// TwinCAT 3 PLC project ExamplePlc
// Company: Sensata Technologies Mechanization
// ProgramVersion: 3.1.4023.0
// libraries:
//   Sensata_Common, * (Sensata Technologies)
//   Sensata_PressureTransducers, * (Sensata Technologies)
//   Sensata_Utilities, * (Sensata Technologies)
//   Tc2_Standard, * (Beckhoff Automation GmbH)
//   Tc2_System, * (Beckhoff Automation GmbH)
//   Tc2_Utilities, * (Beckhoff Automation GmbH)
//   Tc3_Module, * (Beckhoff Automation GmbH)
// project tree:
//   0 Program/ PRG_Main.TcPOU
//   1 Module/0 Machines/ FB_ExampleMachine.TcPOU (not stored)
//   1 Module/1 Stations/ FB_ExampleStation.TcPOU (not stored)
//   1 Module/2 Devices/ FB_ExampleDevice.TcPOU (not stored)
//   / TASK_Main.TcTTO (not stored)
// real-time tasks:
//   TASK TASK_Main: cycle T#10ms, priority 20, ADS port 350

// ---- 0 Program/PRG_Main.TcPOU
PROGRAM PRG_Main
VAR
	bTestInput: BOOL;
	bTestOutput: BOOL;
	fbMachine: FB_ExampleMachine;
	fbStation1: FB_ExampleStation;
	fbStation2: FB_ExampleStation;
	fbStation3: FB_ExampleStation;
	fbStation4: FB_ExampleStation;
	bStart: BOOL;
	bAbort: BOOL;
	bReset: BOOL;
	bStop: BOOL;
	bSuspend: BOOL;
	fbDevice1: FB_ExampleDevice;
	fbDevice2: FB_ExampleDevice;
	fbDevice3: FB_ExampleDevice;
	fbDevice4: FB_ExampleDevice;
	bPoweredOn: BOOL;
//	FB_AdsDeviceAPI_0: FB_AdsDeviceAPI;
	FB_AdsDeviceAPI_0 : FB_AdsCommandRouter;
	bConnectToAlicatAbs: BOOL;
	bRes_AlicatAbsConnected: BOOL;
	bTestADSServer: BOOL;
	strTarget: T_MaxString;
	strCommand: T_MaxString;
	arrParams: T_ApiMethodParameters;
	MyResults: T_MaxString;
	bInterfaceTest : BOOL;
	bDisconnectFromAlicatAbs: BOOL;
	bRes_AlicatAbsDisConnected: BOOL;
	bGetPressure: BOOL;
	bGetPressureSuccessful: BOOL;
	bGetAlicatData: BOOL;
	bGetAlicatDataSuccessful: BOOL;
	bLockDisplay: BOOL;
	bLockDisplaySuccessful: BOOL;
	bUnlockDisplay: BOOL;
	bUnlockDisplaySuccessful: BOOL;
	AlicatAbsolutePressureTransducer_1: FB_AbsolutePressureTransducer;
END_VAR

bTestOutput := bTestInput;

A_Machine();
//A_Station1();
//A_Station2();
//A_Station3();
//A_Station4();
//bInterfaceTest := MyLaser1.fbApi.P_bDeviceInterfaceBusy;



IF bConnectToAlicatAbs THEN
	bRes_AlicatAbsConnected := AlicatAbsolutePressureTransducer_1.M_Connect();
	IF bRes_AlicatAbsConnected THEN
		bConnectToAlicatAbs := FALSE;
	ELSIF AlicatAbsolutePressureTransducer_1.P_bError THEN
		bConnectToAlicatAbs := FALSE;
		AlicatAbsolutePressureTransducer_1.M_ClearError();
	END_IF
END_IF

IF bDisconnectFromAlicatAbs THEN
	bRes_AlicatAbsDisConnected := AlicatAbsolutePressureTransducer_1.M_Disconnect();
	IF bRes_AlicatAbsConnected THEN
		bDisconnectFromAlicatAbs := FALSE;
	ELSIF AlicatAbsolutePressureTransducer_1.P_bError THEN
		bDisconnectFromAlicatAbs := FALSE;
		AlicatAbsolutePressureTransducer_1.M_ClearError();
	END_IF
END_IF

IF bGetPressure THEN
	bGetPressureSuccessful := AlicatAbsolutePressureTransducer_1.M_GetPressure();
	IF bGetPressureSuccessful THEN
		bGetPressure := FALSE;
	ELSIF AlicatAbsolutePressureTransducer_1.P_bError THEN
		bGetPressure := FALSE;
		AlicatAbsolutePressureTransducer_1.M_ClearError();
	END_IF
END_IF

IF bGetAlicatData THEN
	bGetAlicatDataSuccessful := AlicatAbsolutePressureTransducer_1.M_GetAlicatData();
	IF bGetAlicatDataSuccessful THEN
		bGetAlicatData := FALSE;
	ELSIF AlicatAbsolutePressureTransducer_1.P_bError THEN
		bGetAlicatData := FALSE;
		AlicatAbsolutePressureTransducer_1.M_ClearError();
	END_IF
END_IF

IF bLockDisplay THEN
	bLockDisplaySuccessful := AlicatAbsolutePressureTransducer_1.M_LockDisplay();
	IF bLockDisplaySuccessful THEN
		bLockDisplay := FALSE;
	ELSIF AlicatAbsolutePressureTransducer_1.P_bError THEN
		bLockDisplay := FALSE;
		AlicatAbsolutePressureTransducer_1.M_ClearError();
	END_IF
END_IF

IF bUnlockDisplay THEN
	bUnlockDisplaySuccessful := AlicatAbsolutePressureTransducer_1.M_UnlockDisplay();
	IF bUnlockDisplaySuccessful THEN
		bUnlockDisplay := FALSE;
	ELSIF AlicatAbsolutePressureTransducer_1.P_bError THEN
		bUnlockDisplay := FALSE;
		AlicatAbsolutePressureTransducer_1.M_ClearError();
	END_IF
END_IF


//IF bConnectToLaserMarker THEN
//	bRes_LaserConnected := MyLaser1.M_Connect();
//	IF bRes_LaserConnected THEN
//	//Add some timer based logic to do error handling.
//		bConnectToLaserMarker := FALSE;
//	ELSIF MyLaser1.P_bError THEN
//		bConnectToLaserMarker := FALSE;
//		MyLaser1.M_ClearError();
//	END_IF
//END_IF


//IF bDisconnectFromLaserMarker THEN
//	bRes_LaserDisconnected := MyLaser1.M_Disconnect();
//	IF bRes_LaserDisconnected THEN
//		bDisconnectFromLaserMarker := FALSE;
//	ELSIF MyLaser1.P_bError THEN
//		bDisconnectFromLaserMarker := FALSE;
//		MyLaser1.M_ClearError();
//	END_IF
//END_IF


//IF bPeakCurrentProgramInLaser THEN
//	bRes_PeakCurrentProgramInLaser := MyLaser1.M_PeakCurrentProgram();
//	IF bRes_PeakCurrentProgramInLaser THEN
//		bPeakCurrentProgramInLaser := FALSE;
//	ELSIF MyLaser1.P_bError THEN
//		bPeakCurrentProgramInLaser := FALSE;
//		MyLaser1.M_ClearError();
//	END_IF
//END_IF


//IF bSendProgramToLaser THEN
//	bRes_SendProgramtoLaser := MyLaser1.M_SendProgramtoLaser(filepath,LaserMemoryLocation);
//	IF bRes_SendProgramtoLaser THEN
//		bSendProgramToLaser := FALSE;
//	ELSIF MyLaser1.P_bError THEN
//		bSendProgramToLaser := FALSE;
//		MyLaser1.M_ClearError();
//	END_IF
//END_IF

//IF bSaveCurrentLaserProgramtoPC THEN
//	bRes_SaveCurrentLaserProgramtoPC := MyLaser1.M_SaveCurrentLaserProgramtoPC(LaserProgramFolderPath, out_bool_SaveProgramToPC_Success => SaveCurrentLaserProgramToPCSuccess);
//	IF bRes_SaveCurrentLaserProgramtoPC THEN
////		SaveCurrentLaserProgramToPCSuccess := MyLaser1
//		bSaveCurrentLaserProgramtoPC := FALSE;
//	ELSIF MyLaser1.P_bError THEN
//		bSaveCurrentLaserProgramtoPC := FALSE;
//		MyLaser1.M_ClearError();
//	END_IF
//END_IF

//IF bStartMarking THEN
//	bRes_StartMarking := MyLaser1.M_StartMarking();
//	IF bRes_StartMarking THEN
//		bStartMarking := FALSE;
//	ELSIF MyLaser1.P_bError THEN
//		bStartMarking := FALSE;
//		MyLaser1.M_ClearError();
//	END_IF
//END_IF

//IF bStopMarking THEN
//	bRes_StopMarking := MyLaser1.M_StopMarking();
//	IF bRes_StopMarking THEN
//		bStopMarking := FALSE;
//	ELSIF MyLaser1.P_bError THEN
//		bStopMarking := FALSE;
//		MyLaser1.M_ClearError();
//	END_IF
//END_IF

//IF bClearLaserErrors THEN
//	bRes_ClearLaserErrors := MyLaser1.M_ClearLaserErrors();
//	IF bRes_ClearLaserErrors THEN
//		bClearLaserErrors := FALSE;
//	ELSIF MyLaser1.P_bError THEN
//		bClearLaserErrors := FALSE;
//		MyLaser1.M_ClearError();
//	END_IF
//END_IF

//IF bResetErrors THEN
//	bRes_Reset := MyLaser1.M_Reset();
//	IF bRes_Reset THEN
//		bResetErrors := FALSE;
//	ELSIF MyLaser1.P_bError THEN
//		bResetErrors := FALSE;
//		MyLaser1.M_ClearError();
//	END_IF
//END_IF

//IF bUpdateProgramBlockInTheLaser THEN
//	bRes_UpdateProgramBlockInTheLaser := MyLaser1.M_UpdateSingleProgramBlockData(LaserMemoryLocation, _blockNumber, _blockData, _blockType, out_bool_UpdateData_Success => _bUpdateSingleBlockDataSuccess);
//	IF bRes_UpdateProgramBlockInTheLaser THEN
//		bUpdateProgramBlockInTheLaser := FALSE;
//	ELSIF MyLaser1.P_bError THEN
//		bUpdateProgramBlockInTheLaser := FALSE;
//		MyLaser1.M_ClearError();
//	END_IF
//END_IF

//IF bUpdateProgramBlockMarkEnabledInTheLaser THEN
//	bRes_UpdateProgramBlockMarkEnabledInTheLaser := MyLaser1.M_UpdateSingleProgramBlockMarkEnabled( LaserProgramMemoryLocation := LaserMemoryLocation, BlockNumber := _blockNumber, BlockType := _blockType ,MarkEnabled := _markenabled, out_bool_MarkEnabled_Success => _bUpdateSingleBlockMarkEnabled_Success);
//	IF bRes_UpdateProgramBlockMarkEnabledInTheLaser THEN
//		bUpdateProgramBlockMarkEnabledInTheLaser := FALSE;
//	ELSIF MyLaser1.P_bError THEN
//		bUpdateProgramBlockMarkEnabledInTheLaser := FALSE;
//		MyLaser1.M_ClearError();
//	END_IF
//END_IF

//IF bGetLaserStatus THEN
//	bRes_GetLaserStatus := MyLaser1.M_GetLaserStatus( _out_string_laserStatus => _string_laserstatus);
//	IF bRes_GetLaserStatus THEN
//		bGetLaserStatus := FALSE;
//	ELSIF MyLaser1.P_bError THEN
//		bGetLaserStatus := FALSE;
//		MyLaser1.M_ClearError();
//	END_IF
//END_IF

//IF bGetLaserErrorStatus THEN
//	bRes_GetLaserErrorStatus := MyLaser1.M_GetLaserErrorStatus( out_bool_IsLaserError => _bIsLaserError);
//	IF bRes_GetLaserErrorStatus THEN
//		bGetLaserErrorStatus := FALSE;
//	ELSIF MyLaser1.P_bError THEN
//		bGetLaserErrorStatus := FALSE;
//		MyLaser1.M_ClearError();
//	END_IF
//END_IF

//IF bGetLaserActivatedStatus THEN
//	bRes_GetLaserActivatedStatus := MyLaser1.M_GetLaserActivatedStatus( out_IsLaserActivated => _bIsLaserActivated);
//	IF bRes_GetLaserActivatedStatus THEN
//		bGetLaserActivatedStatus := FALSE;
//	ELSIF MyLaser1.P_bError THEN
//		bGetLaserActivatedStatus := FALSE;
//		MyLaser1.M_ClearError();
//	END_IF
//END_IF

//IF bGetLaserMarkingStatus THEN
//	bRes_GetLaserMarkingStatus := MyLaser1.M_GetLaserMarkingStatus( out_bool_IsLaserMarking => _bIsLaserMarking);
//	IF bRes_GetLaserMarkingStatus THEN
//		bGetLaserMarkingStatus := FALSE;
//	ELSIF MyLaser1.P_bError THEN
//		bGetLaserMarkingStatus := FALSE;
//		MyLaser1.M_ClearError();
//	END_IF
//END_IF

ACTION A_Machine:
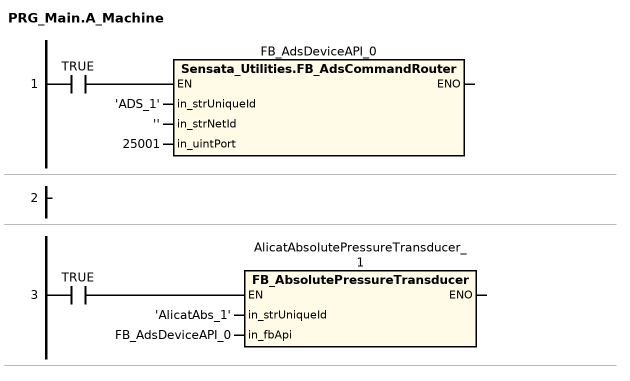
// NETWORK 1
FB_AdsDeviceAPI_0(in_strUniqueId := 'ADS_1', in_strNetId := '', in_uintPort := 25001); // Sensata_Utilities.FB_AdsCommandRouter

// NETWORK 2

// NETWORK 3
AlicatAbsolutePressureTransducer_1(in_strUniqueId := 'AlicatAbs_1', in_fbApi := FB_AdsDeviceAPI_0); // FB_AbsolutePressureTransducer
END_ACTION

ACTION A_Station1:
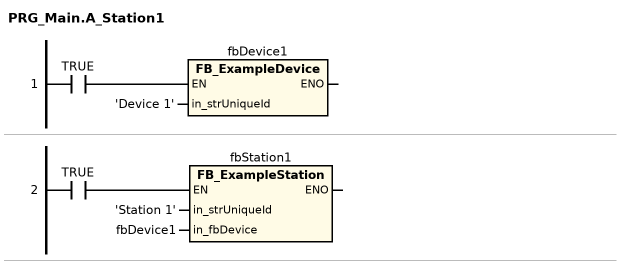
// NETWORK 1
fbDevice1(in_strUniqueId := 'Device 1'); // FB_ExampleDevice

// NETWORK 2
fbStation1(in_strUniqueId := 'Station 1', in_fbDevice := fbDevice1); // FB_ExampleStation
END_ACTION

ACTION A_Station2:
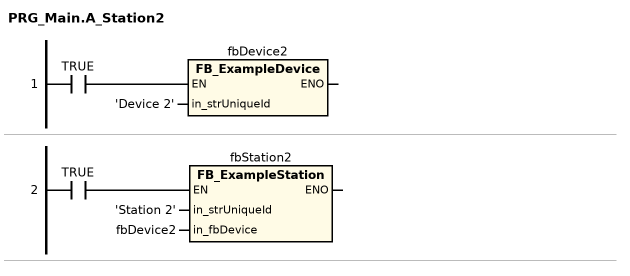
// NETWORK 1
fbDevice2(in_strUniqueId := 'Device 2'); // FB_ExampleDevice

// NETWORK 2
fbStation2(in_strUniqueId := 'Station 2', in_fbDevice := fbDevice2); // FB_ExampleStation
END_ACTION

ACTION A_Station3:
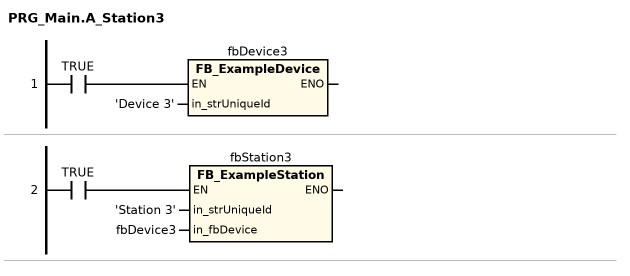
// NETWORK 1
fbDevice3(in_strUniqueId := 'Device 3'); // FB_ExampleDevice

// NETWORK 2
fbStation3(in_strUniqueId := 'Station 3', in_fbDevice := fbDevice3); // FB_ExampleStation
END_ACTION

ACTION A_Station4:
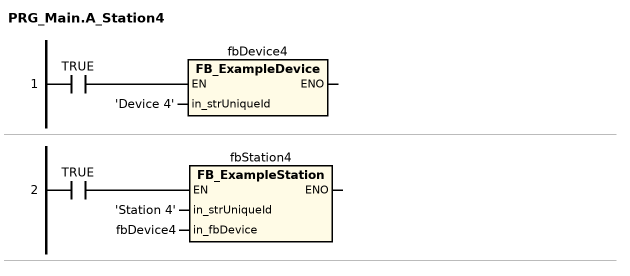
// NETWORK 1
fbDevice4(in_strUniqueId := 'Device 4'); // FB_ExampleDevice

// NETWORK 2
fbStation4(in_strUniqueId := 'Station 4', in_fbDevice := fbDevice4); // FB_ExampleStation
END_ACTION

END_PROGRAM
